INTERFACE I_ParameterAddedEvent EXTENDS I_Event

PROPERTY PUBLIC TargetParameter : I_Parameter
GET
END_GET
END_PROPERTY

END_INTERFACE

(* stored: Version 1.1.0.1, ProductVersion 3.1.4024.12
   Itf I_ParameterAddedEvent: Id {a3faac56-0276-00b7-261f-860c5e2f1a5b}
   Property TargetParameter: Id {b61a6fcc-773b-0407-0b40-1d71dbdd1f81}
   Get Get: Id {11f1107e-7725-0c49-07ff-064b847ff161} *)
